// TIA Portal project "PLC_Mixing_system" (V18)

(* hardware
DEVICE "S7-1200 station_2"  S7-1200 Station
   slot 0: "Rack_0"  S7-1200 Rack  Rack  V1.0
   slot 1: "PLC"  CPU 1215C DC/DC/Rly  6ES7 215-1HG40-0XB0  V4.6
*)

// ===== PLC "PLC"  CPU 1215C DC/DC/Rly =====

VAR_GLOBAL   // PLC tag table "Default tag table"
   "L_LEVEL" AT %I0.0 : Bool;
   "H_LEVEL" AT %I0.1 : Bool;
   "STOP" AT %I0.2 : Bool;
   "PUMP_1" AT %Q0.0 : Bool;
   "PUMP_2" AT %Q0.1 : Bool;
   "VALVE" AT %Q0.2 : Bool;
   "MIXER" AT %Q0.3 : Bool;
   "Tag_2" AT %M0.0 : Bool;
   "Tag_1" AT %M0.1 : Bool;
   "Tag_3" AT %M0.2 : Bool;
END_VAR

// folder: System blocks/Program resources

DATA_BLOCK "Timer_0_DB"   // DB1
{ S7_Optimized_Access := 'TRUE' }
AUTHOR : Simatic
FAMILY : IEC
NAME : IEC_TMR
VERSION : 1.0
// stored: InstanceOfName IEC_TIMER
"IEC_TIMER"
BEGIN
END_DATA_BLOCK

// folder: (top level)

ORGANIZATION_BLOCK "Main"   // OB1, LAD, ProgramCycle
TITLE = "Main Program Sweep (Cycle)"
{ S7_Optimized_Access := 'TRUE' }
VERSION : 0.1
BEGIN

REGION Network 1
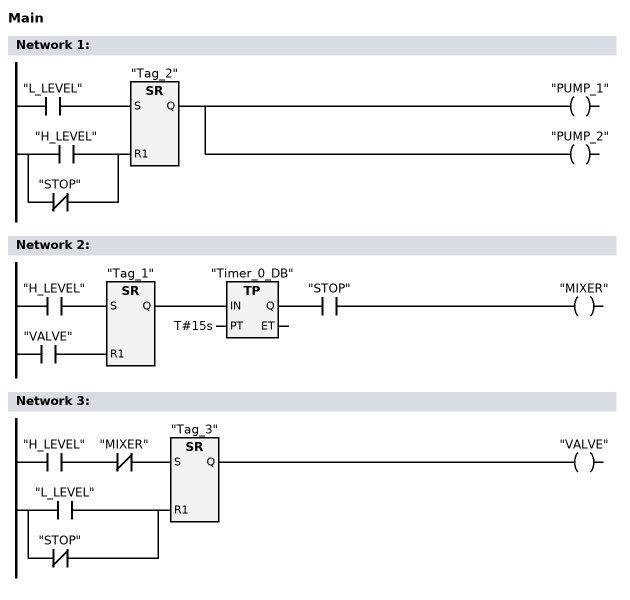
   RUNG wire#powerrail
      Contact( "L_LEVEL" )
      S_SR(operand := "Tag_2", r1 := wire#w1)
      wire#w2
      Coil( "PUMP_1" )
   END_RUNG
   RUNG wire#powerrail
      Contact( "H_LEVEL" )
   END_RUNG wire#w1
   RUNG wire#powerrail
      I_Contact( "STOP" )
   END_RUNG wire#w1
   RUNG wire#w2
      Coil( "PUMP_2" )
   END_RUNG
   // the same network as SCL:
   IF "L_LEVEL" THEN
       "Tag_2" := TRUE;   // SR flip-flop
   END_IF;
   IF "H_LEVEL" OR NOT "STOP" THEN "Tag_2" := FALSE; END_IF;
   "PUMP_1" := "Tag_2";
   "PUMP_2" := "Tag_2";
END_REGION

REGION Network 2
   IF "H_LEVEL" THEN
       "Tag_1" := TRUE;   // SR flip-flop
   END_IF;
   IF "VALVE" THEN "Tag_1" := FALSE; END_IF;
   "Timer_0_DB".TP(IN := "Tag_1", PT := T#15s);
   "MIXER" := "Timer_0_DB".Q AND "STOP";
END_REGION

REGION Network 3
   RUNG wire#powerrail
      Contact( "H_LEVEL" )
      I_Contact( "MIXER" )
      S_SR(operand := "Tag_3", r1 := wire#w1)
      Coil( "VALVE" )
   END_RUNG
   RUNG wire#powerrail
      Contact( "L_LEVEL" )
   END_RUNG wire#w1
   RUNG wire#powerrail
      I_Contact( "STOP" )
   END_RUNG wire#w1
   // the same network as SCL:
   IF "H_LEVEL" AND NOT "MIXER" THEN
       "Tag_3" := TRUE;   // SR flip-flop
   END_IF;
   IF "L_LEVEL" OR NOT "STOP" THEN "Tag_3" := FALSE; END_IF;
   "VALVE" := "Tag_3";
END_REGION
END_ORGANIZATION_BLOCK

ORGANIZATION_BLOCK "Main_SCL"   // OB123, SCL, ProgramCycle
TITLE = "Main Program Sweep (Cycle)"
{ S7_Optimized_Access := 'TRUE' }
VERSION : 0.1
   VAR_INPUT
      Initial_Call : Bool;   // Initial call of this OB
      Remanence : Bool;   // =True, if remanent data are available
   END_VAR
BEGIN
   REGION VAR

   END_REGION
END_ORGANIZATION_BLOCK